PROGRAM MAIN
VAR
END_VAR

END_PROGRAM

(* stored: Version 1.1.0.1
   POU MAIN: Id {d28f26a4-102d-413e-a996-ee61b6348cd0} *)
